PROGRAM MAIN
VAR
END_VAR

END_PROGRAM

(* stored: Version 1.1.0.1
   POU MAIN: Id {6e098e0f-bd53-48df-96f2-483c0c7bd17e} *)
